TYPE ST_Shaker :
STRUCT
	
q_xPwrDO	:	BOOL;
xIlk		:	BOOL;
i_xSwitch	:	BOOL;
i_xEpics	:	BOOL;

END_STRUCT
END_TYPE

(* stored: Version 1.1.0.1, ProductVersion 3.1.0.24
   DUT ST_Shaker: Id {91397fcc-47b0-4fa6-90e4-4877149b614d} *)
